// TIA Portal V19 export
DATA_BLOCK "Area01_HU"   // DB59
// stored: InstanceOfName Area01_HU_FB, InstanceOfType FB
"Area01_HU_FB"
   // VAR_INPUT
   //    AreaInterface : "AreaInterface";
   // END_VAR
   // VAR_OUTPUT
   //    MachineInterface : "MachineInterface";
   // END_VAR
   // VAR
   //    Pump : "HU_Pump";
   //    Tank { S7_SetPoint := 'True'} : "HU_Tank";
   //    HMI : Struct
   //       Pressure_CoilCar : Real;
   //       Pressure_Peeler : Real;
   //       Pressure_JB_Cut : Real;
   //    END_STRUCT;
   // END_VAR
BEGIN
END_DATA_BLOCK
